PROGRAM MAIN
VAR
	aStructs:ARRAY[1..20] OF st01;
	
END_VAR

prgFileHnd();
prgFileManipulation();

END_PROGRAM

(* stored: Version 1.1.0.1, ProductVersion 3.1.4024.12
   POU MAIN: Id {092db28a-b308-4dc7-9e44-1fe289d730d9}, SpecialFunc None *)
